Yaskawa INFORM job: H_profile_cylinder_program.JBI

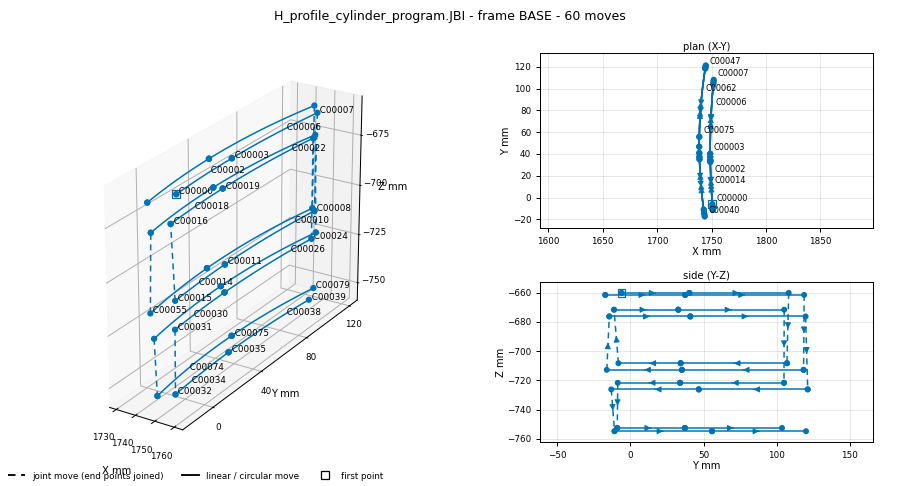
[picture p0: tool path of H_profile_cylinder_program.JBI in frame BASE, 60 of 85 moves have a stored position in this frame; points joined in program order, loops and branches not executed]
/JOB
//NAME H_profile_cylinder_program
//POS
///NPOS 80,0,80,0,0,0
///TOOL 0
///POSTYPE BASE
///RECTAN
///RCONF 0,0,0,0,0,0,0,0,0,0,0,0,0,0,0,0,0,0,0,0,0,0,0,0
C00000=1750.776366,-6.143910,-660.203500,-175.000000,-90.000000,5.000000
C00001=1750.776366,-6.143910,-660.203500,-175.000000,-90.000000,5.000000
C00002=1749.262674,20.355006,-660.203500,-175.000000,-90.000000,5.000000
C00003=1748.845326,40.236114,-660.203500,-175.000000,-89.999999,5.000000
C00004=1748.845326,40.236114,-660.203500,-175.000000,-89.999999,5.000000
C00005=1748.845326,40.236114,-660.203500,-175.000000,-89.999999,5.000000
C00006=1749.954705,81.740852,-660.203500,175.000000,-90.000000,5.000000
C00007=1752.060497,108.150080,-660.203500,174.261683,-90.000000,5.000000
C00008=1751.945212,106.992309,-708.247000,174.365265,-90.000000,5.000000
C00009=1751.945212,106.992309,-708.247000,174.365265,-90.000000,5.000000
C00010=1750.421001,88.949367,-708.247000,175.000000,-90.000000,5.000000
C00011=1748.905843,34.282795,-708.247000,-175.000000,-90.000000,5.000000
C00012=1748.905843,34.282795,-708.247000,-175.000000,-90.000000,5.000000
C00013=1748.905843,34.282795,-708.247000,-175.000000,-90.000000,5.000000
C00014=1749.733423,9.815421,-708.247000,-175.000000,-89.999999,5.000000
C00015=1750.944732,-8.261716,-708.247000,-175.000000,-90.000000,5.000000
C00016=1751.193451,-11.240410,-671.664460,-175.000000,-60.000000,5.000000
C00017=1751.193451,-11.240410,-671.664460,-175.000000,-60.000000,5.000000
C00018=1749.877681,7.189227,-671.664460,175.000000,-60.000000,5.000000
C00019=1748.931483,32.683652,-671.664460,-175.000000,-60.000000,5.000000
C00020=1748.931483,32.683652,-671.664460,-175.000000,-60.000000,5.000000
C00021=1748.931483,32.683652,-671.664460,-175.000000,-60.000000,5.000000
C00022=1750.213187,85.890163,-671.664460,175.000000,-60.000000,-5.000000
C00023=1751.757324,105.058088,-671.664460,175.000000,-60.000000,-5.461728
C00024=1751.746407,104.943804,-721.641960,-175.000000,-60.000000,-5.451508
C00025=1751.746407,104.943804,-721.641960,-175.000000,-60.000000,-5.451508
C00026=1750.258716,86.579202,-721.641960,-175.000000,-60.000000,-5.000000
C00027=1748.911657,33.897521,-721.641960,175.000000,-60.000000,5.000000
C00028=1748.911657,33.897521,-721.641960,175.000000,-60.000000,5.000000
C00029=1748.911657,33.897521,-721.641960,175.000000,-60.000000,5.000000
C00030=1749.983366,5.379340,-721.641960,175.000000,-60.000000,5.000000
C00031=1750.981390,-8.711427,-721.641960,175.000000,-60.000000,5.000000
C00032=1751.007408,-9.028273,-752.523460,175.000000,-60.000000,5.000000
C00033=1751.007408,-9.028273,-752.523460,175.000000,-60.000000,5.000000
C00034=1750.149075,2.702211,-752.523460,-175.000000,-60.000000,5.000000
C00035=1748.869570,37.174327,-752.523460,175.000000,-60.000000,5.000000
C00036=1748.869570,37.174327,-752.523460,175.000000,-60.000000,5.000000
C00037=1748.869570,37.174327,-752.523460,175.000000,-60.000000,5.000000
C00038=1750.064811,83.561514,-752.523460,-175.000000,-60.000000,-5.000000
C00039=1751.616507,103.567029,-752.523460,175.000000,-60.000000,-5.328394
C00040=1743.761471,-17.233943,-661.559500,-171.361988,-90.000000,5.000000
C00041=1743.761471,-17.233943,-661.559500,-171.361988,-90.000000,5.000000
C00042=1740.743449,7.217821,-661.559500,-174.565428,-90.000000,5.000000
C00043=1738.914210,37.392395,-661.559500,-175.000000,-90.000000,5.000000
C00044=1738.914210,37.392395,-661.559500,-175.000000,-90.000000,5.000000
C00045=1738.914210,37.392395,-661.559500,-175.000000,-90.000000,5.000000
C00046=1740.204972,84.585956,-661.559500,175.000000,-89.999999,5.000000
C00047=1744.320922,118.731878,-661.559500,170.890487,-90.000000,5.000000
C00048=1744.258093,118.338904,-712.780500,170.942225,-90.000000,5.000000
C00049=1744.258093,118.338904,-712.780500,170.942225,-90.000000,5.000000
C00050=1740.276955,85.462590,-712.780500,175.000000,-90.000000,5.000000
C00051=1738.978438,35.161072,-712.780500,-175.000000,-90.000000,5.000000
C00052=1738.978438,35.161072,-712.780500,-175.000000,-90.000000,5.000000
C00053=1738.978438,35.161072,-712.780500,-175.000000,-90.000000,5.000000
C00054=1741.293892,1.788721,-712.780500,-173.855984,-89.999999,5.000000
C00055=1743.605509,-16.199025,-712.780500,-171.498054,-89.999999,5.000000
C00056=1743.354904,-14.499939,-676.254960,-175.000000,-60.000000,8.278663
C00057=1743.354904,-14.499939,-676.254960,-175.000000,-60.000000,8.278663
C00058=1740.744634,7.205366,-676.254960,175.000000,-60.000000,5.436198
C00059=1738.836002,40.905586,-676.254960,175.000000,-60.000000,5.000000
C00060=1738.836002,40.905586,-676.254960,175.000000,-60.000000,5.000000
C00061=1738.836002,40.905586,-676.254960,175.000000,-60.000000,5.000000
C00062=1741.110272,94.387748,-676.254960,175.000000,-60.000000,-5.916786
C00063=1744.479860,119.715987,-676.254960,175.000000,-60.000000,-9.239112
C00064=1744.717568,121.162141,-726.145960,-175.000000,-60.000000,-9.429645
C00065=1744.717568,121.162141,-726.145960,-175.000000,-60.000000,-9.429645
C00066=1741.508512,98.078742,-726.145960,175.000000,-60.000000,-6.399427
C00067=1738.768135,46.717682,-726.145960,175.000000,-60.000000,5.000000
C00068=1738.768135,46.717682,-726.145960,175.000000,-60.000000,5.000000
C00069=1738.768135,46.717682,-726.145960,175.000000,-60.000000,5.000000
C00070=1740.435829,10.588510,-726.145960,175.000000,-60.000000,5.000000
C00071=1743.157421,-13.127559,-726.145960,175.000000,-60.000000,8.098407
C00072=1742.848440,-10.915949,-754.724460,175.000000,-60.000000,7.808089
C00073=1742.848440,-10.915949,-754.724460,175.000000,-60.000000,7.808089
C00074=1739.952060,16.597725,-754.724460,175.000000,-60.000000,5.000000
C00075=1738.814674,55.742173,-754.724460,175.000000,-60.000000,-5.000000
C00076=1738.814674,55.742173,-754.724460,175.000000,-60.000000,-5.000000
C00077=1738.814674,55.742173,-754.724460,175.000000,-60.000000,-5.000000
C00078=1742.339629,104.995047,-754.724460,175.000000,-60.000000,-7.305074
C00079=1744.526286,120.000803,-754.724460,175.000000,-60.000000,-9.276629
///POSTYPE PULSE
///PULSE
EX00000=96256.0
EX00001=280576.0
///POSTYPE PULSE
///PULSE
EC00000=96256.0
EC00001=96256.0
EC00002=96256.0
EC00003=96256.0
EC00004=96256.0
EC00005=96256.0
EC00006=96256.0
EC00007=96256.0
EC00008=96256.0
EC00009=96256.0
EC00010=96256.0
EC00011=96256.0
EC00012=96256.0
EC00013=96256.0
EC00014=96256.0
EC00015=96256.0
EC00016=96256.0
EC00017=96256.0
EC00018=96256.0
EC00019=96256.0
EC00020=96256.0
EC00021=96256.0
EC00022=96256.0
EC00023=96256.0
EC00024=96256.0
EC00025=96256.0
EC00026=96256.0
EC00027=96256.0
EC00028=96256.0
EC00029=96256.0
EC00030=96256.0
EC00031=96256.0
EC00032=96256.0
EC00033=96256.0
EC00034=96256.0
EC00035=96256.0
EC00036=96256.0
EC00037=96256.0
EC00038=96256.0
EC00039=96256.0
EC00040=280576.0
EC00041=280576.0
EC00042=280576.0
EC00043=280576.0
EC00044=280576.0
EC00045=280576.0
EC00046=280576.0
EC00047=280576.0
EC00048=280576.0
EC00049=280576.0
EC00050=280576.0
EC00051=280576.0
EC00052=280576.0
EC00053=280576.0
EC00054=280576.0
EC00055=280576.0
EC00056=280576.0
EC00057=280576.0
EC00058=280576.0
EC00059=280576.0
EC00060=280576.0
EC00061=280576.0
EC00062=280576.0
EC00063=280576.0
EC00064=280576.0
EC00065=280576.0
EC00066=280576.0
EC00067=280576.0
EC00068=280576.0
EC00069=280576.0
EC00070=280576.0
EC00071=280576.0
EC00072=280576.0
EC00073=280576.0
EC00074=280576.0
EC00075=280576.0
EC00076=280576.0
EC00077=280576.0
EC00078=280576.0
EC00079=280576.0
//INST
///DATE 2023/08/16 15:49
///ATTR SC,RW,RJ
////FRAME BASE
///GROUP1 RB1,ST1
NOP
MOVJ P009 EX000 VJ=15.00
MOVJ C00000 EC00000 VJ=15.0
CALL JOB:SPYON
MOVC C00001 EC00001 V=150.0
MOVC C00002 EC00002 V=150.0
MOVC C00003 EC00003 V=150.0
MOVJ C00004 EC00004 VJ=15.0
MOVC C00005 EC00005 V=150.0
MOVC C00006 EC00006 V=150.0
MOVC C00007 EC00007 V=150.0
MOVJ C00008 EC00008 VJ=15.0
MOVC C00009 EC00009 V=150.0
MOVC C00010 EC00010 V=150.0
MOVC C00011 EC00011 V=150.0
MOVJ C00012 EC00012 VJ=15.0
MOVC C00013 EC00013 V=150.0
MOVC C00014 EC00014 V=150.0
MOVC C00015 EC00015 V=150.0
MOVJ C00016 EC00016 VJ=15.0
MOVC C00017 EC00017 V=150.0
MOVC C00018 EC00018 V=150.0
MOVC C00019 EC00019 V=150.0
MOVJ C00020 EC00020 VJ=15.0
MOVC C00021 EC00021 V=150.0
MOVC C00022 EC00022 V=150.0
MOVC C00023 EC00023 V=150.0
MOVJ C00024 EC00024 VJ=15.0
MOVC C00025 EC00025 V=150.0
MOVC C00026 EC00026 V=150.0
MOVC C00027 EC00027 V=150.0
MOVJ C00028 EC00028 VJ=15.0
MOVC C00029 EC00029 V=150.0
MOVC C00030 EC00030 V=150.0
MOVC C00031 EC00031 V=150.0
MOVJ C00032 EC00032 VJ=15.0
MOVC C00033 EC00033 V=150.0
MOVC C00034 EC00034 V=150.0
MOVC C00035 EC00035 V=150.0
MOVJ C00036 EC00036 VJ=15.0
MOVC C00037 EC00037 V=150.0
MOVC C00038 EC00038 V=150.0
MOVC C00039 EC00039 V=150.0
CALL JOB:SPYOF
MOVJ P009 VJ=15.00
MOVL P009 EX00000 V=150.0
MOVJ C00040 EC00040 VJ=15.0
CALL JOB:SPYON
MOVC C00041 EC00041 V=150.0
MOVC C00042 EC00042 V=150.0
MOVC C00043 EC00043 V=150.0
MOVJ C00044 EC00044 VJ=15.0
MOVC C00045 EC00045 V=150.0
MOVC C00046 EC00046 V=150.0
MOVC C00047 EC00047 V=150.0
MOVJ C00048 EC00048 VJ=15.0
MOVC C00049 EC00049 V=150.0
MOVC C00050 EC00050 V=150.0
MOVC C00051 EC00051 V=150.0
MOVJ C00052 EC00052 VJ=15.0
MOVC C00053 EC00053 V=150.0
MOVC C00054 EC00054 V=150.0
MOVC C00055 EC00055 V=150.0
MOVJ C00056 EC00056 VJ=15.0
MOVC C00057 EC00057 V=150.0
MOVC C00058 EC00058 V=150.0
MOVC C00059 EC00059 V=150.0
MOVJ C00060 EC00060 VJ=15.0
MOVC C00061 EC00061 V=150.0
MOVC C00062 EC00062 V=150.0
MOVC C00063 EC00063 V=150.0
MOVJ C00064 EC00064 VJ=15.0
MOVC C00065 EC00065 V=150.0
MOVC C00066 EC00066 V=150.0
MOVC C00067 EC00067 V=150.0
MOVJ C00068 EC00068 VJ=15.0
MOVC C00069 EC00069 V=150.0
MOVC C00070 EC00070 V=150.0
MOVC C00071 EC00071 V=150.0
MOVJ C00072 EC00072 VJ=15.0
MOVC C00073 EC00073 V=150.0
MOVC C00074 EC00074 V=150.0
MOVC C00075 EC00075 V=150.0
MOVJ C00076 EC00076 VJ=15.0
MOVC C00077 EC00077 V=150.0
MOVC C00078 EC00078 V=150.0
MOVC C00079 EC00079 V=150.0
CALL JOB:SPYOF
MOVJ P009 VJ=15.00
MOVL P009 EX00001 V=150.0
END
